{attribute 'GeneratedUsingTerminal: EL5151-0090-0016'}
{attribute addProperty BoxType "EL5151-0090-0016"}
{attribute addProperty Id "ENC_Status_compactAT %I*ENC_Status_compact_B353648514ENC_Control_compactAT %Q*ENC_Control_compact_21E2D14D6WcStateAT %I*WcState_9091E0EB2InfoDataAT %I*InfoData_32EB74EA10"}
{attribute addProperty CRC "2283980759"}
{attribute addProperty Size "32"}
TYPE EL5151_8822C7D7 :
STRUCT
	{attribute addProperty Name "ENC_Status_compact"}
	ENC_Status_compact : ENC_Status_compact_B3536485;
	{attribute addProperty Name "ENC_Control_compact"}
	ENC_Control_compact : ENC_Control_compact_21E2D14D;
	{attribute addProperty Name "WcState"}
	WcState : WcState_9091E0EB;
	{attribute addProperty Name "InfoData"}
	InfoData : InfoData_32EB74EA;
END_STRUCT
END_TYPE

(* stored: Version 1.2.0.0, ProductVersion 3.1.4024.9
   DUT EL5151_8822C7D7: Id {ad2b6364-0086-41f3-ad30-fe6dbab4b457} *)
